TYPE System_Settings_DUT :
STRUCT
	VTD_Count:  UINT;
	Level_Count:  UINT;
	Cnv_Count:  UInt;
	Shuttle_Count:  UInt;
	Shuttle_Interlock_Timeout:  UINT;
END_STRUCT
END_TYPE

(* stored: Version 1.1.0.1
   DUT System_Settings_DUT: Id {cfee05c6-6b1a-4eb0-8a3b-2315771b5c97} *)
